// TIA Portal project "Project1" (V16)

(* hardware
DEVICE "S7-1200 station_1"  S7-1200 Station
   slot 0: "Rack_0"  S7-1200 Rack  Rack  V1.0
   slot 1: "PLC_1"  CPU 1214C AC/DC/Rly  6ES7 214-1BG40-0XB0  V4.4
DEVICE "PC-System_1"  SIMATIC PC station
   slot 0: "SIMATIC PC station"  Rail  SIMATIC PC-Station  V1.0
      slot 125: "Stationmanager"  Station_Manager  V6.0.4
   slot 1: "HMI_RT_1"  WinCC RT Advanced  6AV2 104-0xxxx-xxxx  16.0.0.0
      slot 33792: "Computer interface"  Host interface
   slot 2: "IE general_1"  IE General  IE_CP  V8.2.0
*)

// ===== PLC "PLC_1"  CPU 1214C AC/DC/Rly =====

VAR_GLOBAL   // PLC tag table "Default tag table"
   "Tag_1" AT %MW20 : UInt;
   "TIMER_1" AT %MW22 : UInt;
   "TIMER_2" AT %MW24 : UInt;
   "INPUT_X1_INT" AT %MW26 : UInt;
   "INPUT_V1_INT" AT %MW28 : UInt;
   "INPUT_X2_INT" AT %MW30 : UInt;
   "INPUT_V2_INT" AT %MW32 : UInt;
   "INPUT_XV1_INT" AT %MW34 : UInt;
   "INPUT_XV2_INT" AT %MW36 : UInt;
   "INPUT_SUM_INT" AT %MW38 : UInt;
   "INPUT_X1" AT %MD50 : Time;
   "INPUT_V1" AT %MD54 : Time;
   "INPUT_XV1" AT %MD58 : Time;
   "INPUT_X2" AT %MD62 : Time;
   "INPUT_V2" AT %MD66 : Time;
   "INPUT_XV2" AT %MD70 : Time;
   "INPUT_SUM" AT %MD78 : Time;
   "Tag_2" AT %MW100 : UInt;
   "Tag_3" AT %MW102 : UInt;
   "Tag_4" AT %MW104 : UInt;
   "Tag_5" AT %MW106 : UInt;
   "Tag_6" AT %MW108 : UInt;
   "X1_TG" AT %MW200 : UInt;
   "V1_TG" AT %MW202 : UInt;
   "X2_TG" AT %MW204 : UInt;
   "V2_TG" AT %MW206 : UInt;
   "XV1_TG" AT %MW208 : UInt;
   "XV2_TG" AT %MW210 : UInt;
   "XV1X2_TG" AT %MW212 : UInt;
   "INPUT_XV1X2_INT" AT %MW40 : UInt;
   "INPUT_XV1X2" AT %MD74 : Time;
   "SUM_TG" AT %MW214 : UInt;
   "Tag_7" AT %M10.0 : Bool;
   "System_Byte" AT %MB1 : Byte;
   "FirstScan" AT %M1.0 : Bool;
   "DiagStatusUpdate" AT %M1.1 : Bool;
   "AlwaysTRUE" AT %M1.2 : Bool;
   "AlwaysFALSE" AT %M1.3 : Bool;
   "Clock_Byte" AT %MB0 : Byte;
   "Clock_10Hz" AT %M0.0 : Bool;
   "Clock_5Hz" AT %M0.1 : Bool;
   "Clock_2.5Hz" AT %M0.2 : Bool;
   "Clock_2Hz" AT %M0.3 : Bool;
   "Clock_1.25Hz" AT %M0.4 : Bool;
   "Clock_1Hz" AT %M0.5 : Bool;
   "Clock_0.625Hz" AT %M0.6 : Bool;
   "Clock_0.5Hz" AT %M0.7 : Bool;
   "Start" AT %M20.0 : Bool;
   "Stop" AT %M20.1 : Bool;
   "Data" AT %MW70 : Int;
   "Tag_8" AT %MW50 : Int;
   "Tag_9" AT %MD10 : Real;
   "Tag_10" AT %MD14 : Real;
   "He_so_k" AT %MD200 : Real;
   "Tag_11" AT %M50.0 : Bool;
   "Tag_12" AT %M5.0 : Bool;
END_VAR

VAR_GLOBAL   // PLC tag table "Tag table_1"
   "X1_IN" AT %I0.0 : Bool;
   "V1_IN" AT %I0.1 : Bool;
   "X2_IN" AT %I0.2 : Bool;
   "V2_IN" AT %I0.3 : Bool;
   "Bus1" AT %MW82 : Int;
   "Car1" AT %MW84 : Int;
   "Motor1" AT %MW86 : Int;
   "Truck1" AT %MW112 : Int;
   "Bus2" AT %MW90 : Int;
   "Car2" AT %MW92 : Int;
   "Motor2" AT %MW94 : Int;
   "Truck2" AT %MW96 : Int;
   "Sum_h1" AT %MW98 : Int;
   "Sum_h2" AT %MW110 : Int;
END_VAR

DATA_BLOCK "DGT"   // DB1
{ S7_Optimized_Access := 'FALSE' }
VERSION : 0.1
   VAR
      RUN : Bool;
      START : Bool;
      STOP : Bool;
      RED_A : Bool;
      YELLOW_A : Bool;
      GREEN_A : Bool;
      RED_B : Bool;
      YELLOW_B : Bool;
      GREEN_B : Bool;
      AUTO : Bool;
      MAN : Bool;
      SETTING : Bool;
      Q_AUTO : Bool;
      Q_MANU : Bool;
      Q_SETTING : Bool;
   END_VAR
BEGIN
END_DATA_BLOCK

DATA_BLOCK "DB_MANU"   // DB7
{ S7_Optimized_Access := 'TRUE' }
VERSION : 0.1
   VAR
      BT_1 : Bool;
      BT_2 : Bool;
      BT_3 : Bool;
   END_VAR
BEGIN
END_DATA_BLOCK

// folder: System blocks/Program resources

DATA_BLOCK "T1"   // DB2
{ S7_Optimized_Access := 'TRUE' }
AUTHOR : Simatic
FAMILY : IEC
NAME : IEC_TMR
VERSION : 1.0
// stored: InstanceOfName IEC_TIMER
"IEC_TIMER"
BEGIN
END_DATA_BLOCK

// folder: (top level)

FUNCTION "MODE_MANU" : Void   // FC1, LAD
{ S7_Optimized_Access := 'TRUE' }
VERSION : 0.1
BEGIN

REGION Network 1
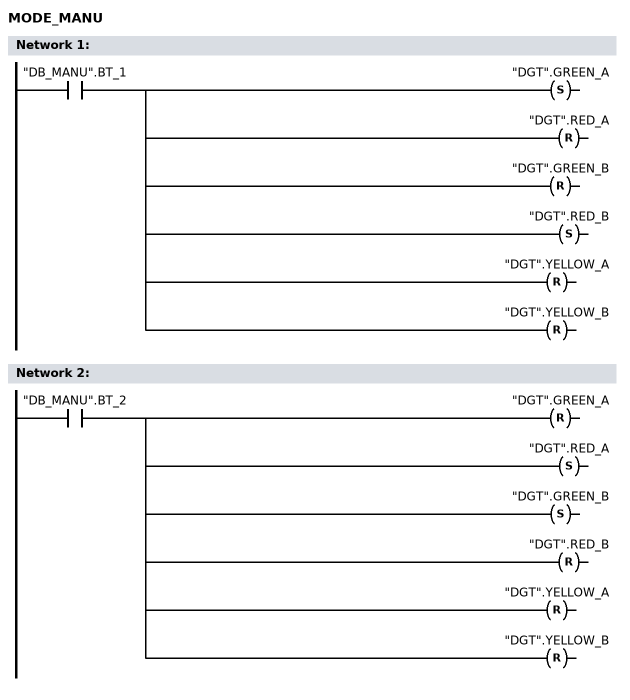
   RUNG wire#powerrail
      Contact( "DB_MANU".BT_1 )
      wire#w1
      S_Coil( "DGT".GREEN_A )
   END_RUNG
   RUNG wire#w1
      R_Coil( "DGT".RED_A )
   END_RUNG
   RUNG wire#w1
      R_Coil( "DGT".GREEN_B )
   END_RUNG
   RUNG wire#w1
      S_Coil( "DGT".RED_B )
   END_RUNG
   RUNG wire#w1
      R_Coil( "DGT".YELLOW_A )
   END_RUNG
   RUNG wire#w1
      R_Coil( "DGT".YELLOW_B )
   END_RUNG
   // the same network as SCL:
   IF "DB_MANU".BT_1 THEN
       "DGT".GREEN_A := TRUE;
       "DGT".RED_A := FALSE;
       "DGT".GREEN_B := FALSE;
       "DGT".RED_B := TRUE;
       "DGT".YELLOW_A := FALSE;
       "DGT".YELLOW_B := FALSE;
   END_IF;
END_REGION

REGION Network 2
   RUNG wire#powerrail
      Contact( "DB_MANU".BT_2 )
      wire#w1
      R_Coil( "DGT".GREEN_A )
   END_RUNG
   RUNG wire#w1
      S_Coil( "DGT".RED_A )
   END_RUNG
   RUNG wire#w1
      S_Coil( "DGT".GREEN_B )
   END_RUNG
   RUNG wire#w1
      R_Coil( "DGT".RED_B )
   END_RUNG
   RUNG wire#w1
      R_Coil( "DGT".YELLOW_A )
   END_RUNG
   RUNG wire#w1
      R_Coil( "DGT".YELLOW_B )
   END_RUNG
   // the same network as SCL:
   IF "DB_MANU".BT_2 THEN
       "DGT".GREEN_A := FALSE;
       "DGT".RED_A := TRUE;
       "DGT".GREEN_B := TRUE;
       "DGT".RED_B := FALSE;
       "DGT".YELLOW_A := FALSE;
       "DGT".YELLOW_B := FALSE;
   END_IF;
END_REGION
END_FUNCTION

FUNCTION "START_UP" : Void   // FC2, LAD
{ S7_Optimized_Access := 'TRUE' }
VERSION : 0.1
BEGIN

REGION Network 1
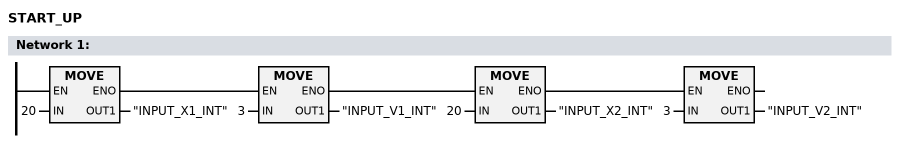
   RUNG wire#powerrail
      Move(in := 20, out1 => "INPUT_X1_INT")
      Move(in := 3, out1 => "INPUT_V1_INT")
      Move(in := 20, out1 => "INPUT_X2_INT")
      Move(in := 3, out1 => "INPUT_V2_INT")
   END_RUNG
   // the same network as SCL:
   "INPUT_X1_INT" := 20;
   "INPUT_V1_INT" := 3;
   "INPUT_X2_INT" := 20;
   "INPUT_V2_INT" := 3;
END_REGION
END_FUNCTION

FUNCTION "MODE_SETTING" : Void   // FC3, LAD
{ S7_Optimized_Access := 'TRUE' }
VERSION : 0.1
   VAR_TEMP   // added for the SCL form of the ladder/FBD networks
      _w1 : Bool;
   END_VAR
BEGIN

REGION Network 1
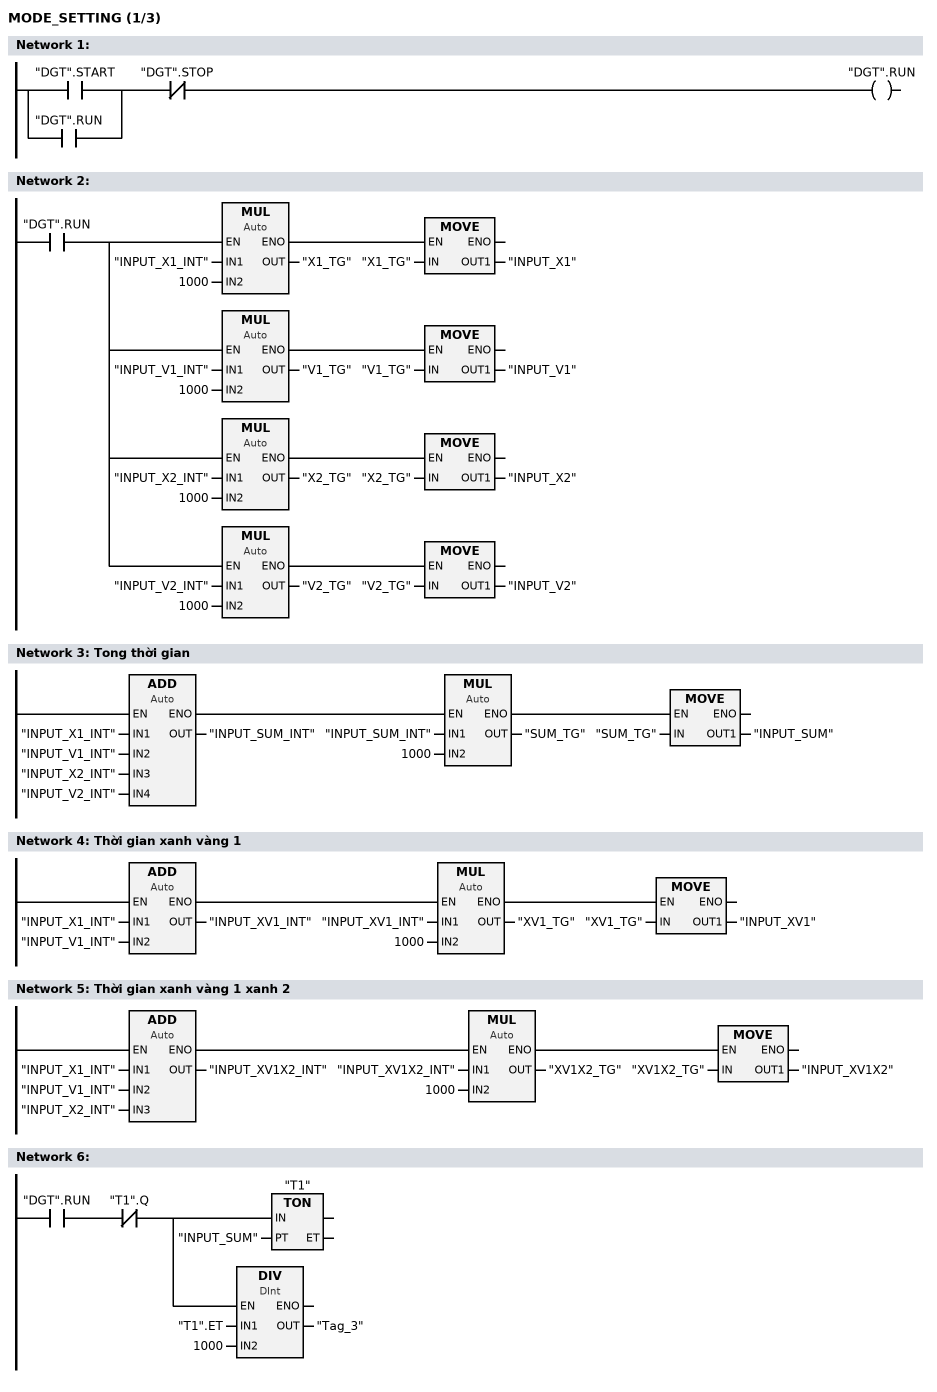
   RUNG wire#powerrail
      Contact( "DGT".START )
      wire#w1
      I_Contact( "DGT".STOP )
      Coil( "DGT".RUN )
   END_RUNG
   RUNG wire#powerrail
      Contact( "DGT".RUN )
   END_RUNG wire#w1
   // the same network as SCL:
   "DGT".RUN := ("DGT".START OR "DGT".RUN) AND NOT "DGT".STOP;
END_REGION

REGION Network 2
   RUNG wire#powerrail
      Contact( "DGT".RUN )
      wire#w1
      Mul(in1 := "INPUT_X1_INT", in2 := 1000, out => "X1_TG")
      Move(in := "X1_TG", out1 => "INPUT_X1")
   END_RUNG
   RUNG wire#w1
      Mul(in1 := "INPUT_V1_INT", in2 := 1000, out => "V1_TG")
      Move(in := "V1_TG", out1 => "INPUT_V1")
   END_RUNG
   RUNG wire#w1
      Mul(in1 := "INPUT_X2_INT", in2 := 1000, out => "X2_TG")
      Move(in := "X2_TG", out1 => "INPUT_X2")
   END_RUNG
   RUNG wire#w1
      Mul(in1 := "INPUT_V2_INT", in2 := 1000, out => "V2_TG")
      Move(in := "V2_TG", out1 => "INPUT_V2")
   END_RUNG
   // the same network as SCL:
   IF "DGT".RUN THEN
       "X1_TG" := "INPUT_X1_INT" * 1000;
       "INPUT_X1" := "X1_TG";
       "V1_TG" := "INPUT_V1_INT" * 1000;
       "INPUT_V1" := "V1_TG";
       "X2_TG" := "INPUT_X2_INT" * 1000;
       "INPUT_X2" := "X2_TG";
       "V2_TG" := "INPUT_V2_INT" * 1000;
       "INPUT_V2" := "V2_TG";
   END_IF;
END_REGION

REGION Network 3: Tong thời gian
   RUNG wire#powerrail
      Add(in1 := "INPUT_X1_INT", in2 := "INPUT_V1_INT", in3 := "INPUT_X2_INT", in4 := "INPUT_V2_INT", out => "INPUT_SUM_INT")
      Mul(in1 := "INPUT_SUM_INT", in2 := 1000, out => "SUM_TG")
      Move(in := "SUM_TG", out1 => "INPUT_SUM")
   END_RUNG
   // the same network as SCL:
   "INPUT_SUM_INT" := "INPUT_X1_INT" + "INPUT_V1_INT" + "INPUT_X2_INT" + "INPUT_V2_INT";
   "SUM_TG" := "INPUT_SUM_INT" * 1000;
   "INPUT_SUM" := "SUM_TG";
END_REGION

REGION Network 4: Thời gian xanh vàng 1
   RUNG wire#powerrail
      Add(in1 := "INPUT_X1_INT", in2 := "INPUT_V1_INT", out => "INPUT_XV1_INT")
      Mul(in1 := "INPUT_XV1_INT", in2 := 1000, out => "XV1_TG")
      Move(in := "XV1_TG", out1 => "INPUT_XV1")
   END_RUNG
   // the same network as SCL:
   "INPUT_XV1_INT" := "INPUT_X1_INT" + "INPUT_V1_INT";
   "XV1_TG" := "INPUT_XV1_INT" * 1000;
   "INPUT_XV1" := "XV1_TG";
END_REGION

REGION Network 5: Thời gian xanh vàng 1 xanh 2
   RUNG wire#powerrail
      Add(in1 := "INPUT_X1_INT", in2 := "INPUT_V1_INT", in3 := "INPUT_X2_INT", out => "INPUT_XV1X2_INT")
      Mul(in1 := "INPUT_XV1X2_INT", in2 := 1000, out => "XV1X2_TG")
      Move(in := "XV1X2_TG", out1 => "INPUT_XV1X2")
   END_RUNG
   // the same network as SCL:
   "INPUT_XV1X2_INT" := "INPUT_X1_INT" + "INPUT_V1_INT" + "INPUT_X2_INT";
   "XV1X2_TG" := "INPUT_XV1X2_INT" * 1000;
   "INPUT_XV1X2" := "XV1X2_TG";
END_REGION

REGION Network 6
   #_w1 := "DGT".RUN AND NOT "T1".Q;
   "T1".TON(IN := #_w1, PT := "INPUT_SUM");
   IF #_w1 THEN "Tag_3" := "T1".ET / 1000; END_IF;
END_REGION

REGION Network 7
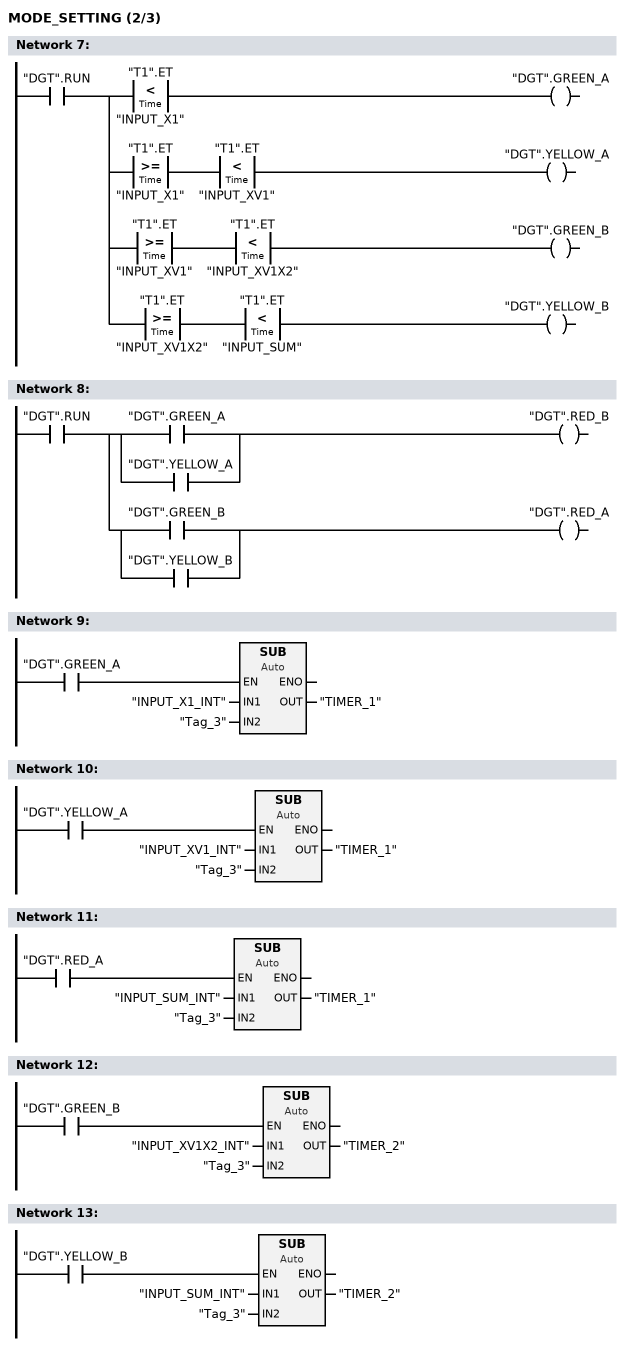
   RUNG wire#powerrail
      Contact( "DGT".RUN )
      wire#w1
      { S7_Templates := "SrcType := Time" } LT_Contact(in1 := "T1".ET, in2 := "INPUT_X1")
      Coil( "DGT".GREEN_A )
   END_RUNG
   RUNG wire#w1
      { S7_Templates := "SrcType := Time" } GE_Contact(in1 := "T1".ET, in2 := "INPUT_X1")
      { S7_Templates := "SrcType := Time" } LT_Contact(in1 := "T1".ET, in2 := "INPUT_XV1")
      Coil( "DGT".YELLOW_A )
   END_RUNG
   RUNG wire#w1
      { S7_Templates := "SrcType := Time" } GE_Contact(in1 := "T1".ET, in2 := "INPUT_XV1")
      { S7_Templates := "SrcType := Time" } LT_Contact(in1 := "T1".ET, in2 := "INPUT_XV1X2")
      Coil( "DGT".GREEN_B )
   END_RUNG
   RUNG wire#w1
      { S7_Templates := "SrcType := Time" } GE_Contact(in1 := "T1".ET, in2 := "INPUT_XV1X2")
      { S7_Templates := "SrcType := Time" } LT_Contact(in1 := "T1".ET, in2 := "INPUT_SUM")
      Coil( "DGT".YELLOW_B )
   END_RUNG
   // the same network as SCL:
   "DGT".GREEN_A := "DGT".RUN AND ("T1".ET < "INPUT_X1");
   "DGT".YELLOW_A := "DGT".RUN AND ("T1".ET >= "INPUT_X1") AND ("T1".ET < "INPUT_XV1");
   "DGT".GREEN_B := "DGT".RUN AND ("T1".ET >= "INPUT_XV1") AND ("T1".ET < "INPUT_XV1X2");
   "DGT".YELLOW_B := "DGT".RUN AND ("T1".ET >= "INPUT_XV1X2") AND ("T1".ET < "INPUT_SUM");
END_REGION

REGION Network 8
   RUNG wire#powerrail
      Contact( "DGT".RUN )
      wire#w1
      Contact( "DGT".GREEN_A )
      wire#w2
      Coil( "DGT".RED_B )
   END_RUNG
   RUNG wire#w1
      Contact( "DGT".YELLOW_A )
   END_RUNG wire#w2
   RUNG wire#w1
      Contact( "DGT".GREEN_B )
      wire#w3
      Coil( "DGT".RED_A )
   END_RUNG
   RUNG wire#w1
      Contact( "DGT".YELLOW_B )
   END_RUNG wire#w3
   // the same network as SCL:
   "DGT".RED_B := "DGT".RUN AND ("DGT".GREEN_A OR "DGT".YELLOW_A);
   "DGT".RED_A := "DGT".RUN AND ("DGT".GREEN_B OR "DGT".YELLOW_B);
END_REGION

REGION Network 9
   RUNG wire#powerrail
      Contact( "DGT".GREEN_A )
      Sub(in1 := "INPUT_X1_INT", in2 := "Tag_3", out => "TIMER_1")
   END_RUNG
   // the same network as SCL:
   IF "DGT".GREEN_A THEN "TIMER_1" := "INPUT_X1_INT" - "Tag_3"; END_IF;
END_REGION

REGION Network 10
   RUNG wire#powerrail
      Contact( "DGT".YELLOW_A )
      Sub(in1 := "INPUT_XV1_INT", in2 := "Tag_3", out => "TIMER_1")
   END_RUNG
   // the same network as SCL:
   IF "DGT".YELLOW_A THEN "TIMER_1" := "INPUT_XV1_INT" - "Tag_3"; END_IF;
END_REGION

REGION Network 11
   RUNG wire#powerrail
      Contact( "DGT".RED_A )
      Sub(in1 := "INPUT_SUM_INT", in2 := "Tag_3", out => "TIMER_1")
   END_RUNG
   // the same network as SCL:
   IF "DGT".RED_A THEN "TIMER_1" := "INPUT_SUM_INT" - "Tag_3"; END_IF;
END_REGION

REGION Network 12
   RUNG wire#powerrail
      Contact( "DGT".GREEN_B )
      Sub(in1 := "INPUT_XV1X2_INT", in2 := "Tag_3", out => "TIMER_2")
   END_RUNG
   // the same network as SCL:
   IF "DGT".GREEN_B THEN "TIMER_2" := "INPUT_XV1X2_INT" - "Tag_3"; END_IF;
END_REGION

REGION Network 13
   RUNG wire#powerrail
      Contact( "DGT".YELLOW_B )
      Sub(in1 := "INPUT_SUM_INT", in2 := "Tag_3", out => "TIMER_2")
   END_RUNG
   // the same network as SCL:
   IF "DGT".YELLOW_B THEN "TIMER_2" := "INPUT_SUM_INT" - "Tag_3"; END_IF;
END_REGION

REGION Network 14
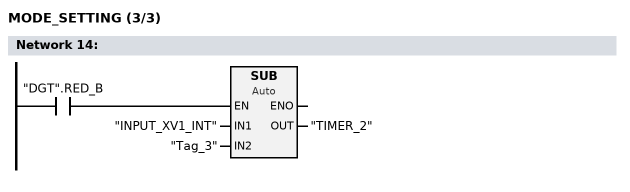
   RUNG wire#powerrail
      Contact( "DGT".RED_B )
      Sub(in1 := "INPUT_XV1_INT", in2 := "Tag_3", out => "TIMER_2")
   END_RUNG
   // the same network as SCL:
   IF "DGT".RED_B THEN "TIMER_2" := "INPUT_XV1_INT" - "Tag_3"; END_IF;
END_REGION
END_FUNCTION

FUNCTION "BROKER" : Void   // FC4, LAD
{ S7_Optimized_Access := 'TRUE' }
VERSION : 0.1
BEGIN

REGION Network 1
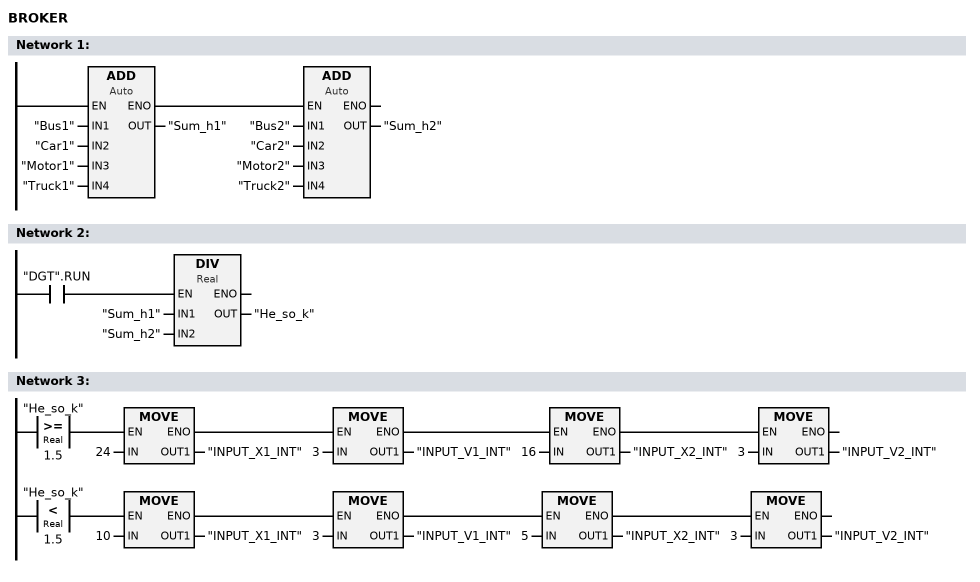
   RUNG wire#powerrail
      Add(in1 := "Bus1", in2 := "Car1", in3 := "Motor1", in4 := "Truck1", out => "Sum_h1")
      Add(in1 := "Bus2", in2 := "Car2", in3 := "Motor2", in4 := "Truck2", out => "Sum_h2")
   END_RUNG
   // the same network as SCL:
   "Sum_h1" := "Bus1" + "Car1" + "Motor1" + "Truck1";
   "Sum_h2" := "Bus2" + "Car2" + "Motor2" + "Truck2";
END_REGION

REGION Network 2
   RUNG wire#powerrail
      Contact( "DGT".RUN )
      { S7_Templates := "SrcType := Real" } Div(in1 := "Sum_h1", in2 := "Sum_h2", out => "He_so_k")
   END_RUNG
   // the same network as SCL:
   IF "DGT".RUN THEN "He_so_k" := "Sum_h1" / "Sum_h2"; END_IF;
END_REGION

REGION Network 3
   RUNG wire#powerrail
      { S7_Templates := "SrcType := Real" } GE_Contact(in1 := "He_so_k", in2 := 1.5)
      Move(in := 24, out1 => "INPUT_X1_INT")
      Move(in := 3, out1 => "INPUT_V1_INT")
      Move(in := 16, out1 => "INPUT_X2_INT")
      Move(in := 3, out1 => "INPUT_V2_INT")
   END_RUNG
   RUNG wire#powerrail
      { S7_Templates := "SrcType := Real" } LT_Contact(in1 := "He_so_k", in2 := 1.5)
      Move(in := 10, out1 => "INPUT_X1_INT")
      Move(in := 3, out1 => "INPUT_V1_INT")
      Move(in := 5, out1 => "INPUT_X2_INT")
      Move(in := 3, out1 => "INPUT_V2_INT")
   END_RUNG
   // the same network as SCL:
   IF "He_so_k" >= 1.5 THEN
       "INPUT_X1_INT" := 24;
       "INPUT_V1_INT" := 3;
       "INPUT_X2_INT" := 16;
       "INPUT_V2_INT" := 3;
   END_IF;
   IF "He_so_k" < 1.5 THEN
       "INPUT_X1_INT" := 10;
       "INPUT_V1_INT" := 3;
       "INPUT_X2_INT" := 5;
       "INPUT_V2_INT" := 3;
   END_IF;
END_REGION
END_FUNCTION

ORGANIZATION_BLOCK "Main"   // OB1, LAD, ProgramCycle
TITLE = "Main Program Sweep (Cycle)"
{ S7_Optimized_Access := 'TRUE' }
VERSION : 0.1
   VAR_INPUT
      Initial_Call : Bool;   // Initial call of this OB
      Remanence : Bool;   // =True, if remanent data are available
   END_VAR
   VAR_TEMP   // added for the SCL form of the ladder/FBD networks
      _w1 : Bool;
   END_VAR
BEGIN

REGION Network 1
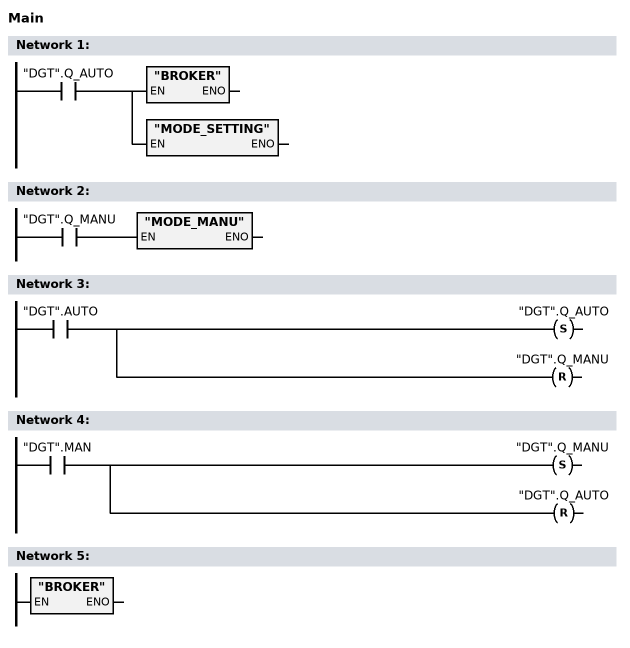
   RUNG wire#powerrail
      Contact( "DGT".Q_AUTO )
      wire#w1
      "BROKER"()
   END_RUNG
   RUNG wire#w1
      "MODE_SETTING"()
   END_RUNG
   // the same network as SCL:
   #_w1 := "DGT".Q_AUTO;
   IF #_w1 THEN
       "BROKER"();
       "MODE_SETTING"();
   END_IF;
END_REGION

REGION Network 2
   RUNG wire#powerrail
      Contact( "DGT".Q_MANU )
      "MODE_MANU"()
   END_RUNG
   // the same network as SCL:
   IF "DGT".Q_MANU THEN "MODE_MANU"(); END_IF;
END_REGION

REGION Network 3
   RUNG wire#powerrail
      Contact( "DGT".AUTO )
      wire#w1
      S_Coil( "DGT".Q_AUTO )
   END_RUNG
   RUNG wire#w1
      R_Coil( "DGT".Q_MANU )
   END_RUNG
   // the same network as SCL:
   IF "DGT".AUTO THEN
       "DGT".Q_AUTO := TRUE;
       "DGT".Q_MANU := FALSE;
   END_IF;
END_REGION

REGION Network 4
   RUNG wire#powerrail
      Contact( "DGT".MAN )
      wire#w1
      S_Coil( "DGT".Q_MANU )
   END_RUNG
   RUNG wire#w1
      R_Coil( "DGT".Q_AUTO )
   END_RUNG
   // the same network as SCL:
   IF "DGT".MAN THEN
       "DGT".Q_MANU := TRUE;
       "DGT".Q_AUTO := FALSE;
   END_IF;
END_REGION

REGION Network 5
   RUNG wire#powerrail
      "BROKER"()
   END_RUNG
   // the same network as SCL:
   "BROKER"();
END_REGION
END_ORGANIZATION_BLOCK

(* ===== HMI "HMI_RT_1" =====
system functions are stored by id; their names below are inferred from use
connection "HMI_Connection_1": ETHERNET, S7_1200_OMS

HMI tags "Default tag table"
   "DGT_XANH_A" : Bool = PLC DGT.GREEN_A AT %DB1.DBX0.5, 1 s
   "DGT_VANG_A" : Bool = PLC DGT.YELLOW_A AT %DB1.DBX0.4, 1 s
   "DGT_DO_A" : Bool = PLC DGT.RED_A AT %DB1.DBX0.3, 1 s
   "INPUT_X1_INT" : UInt = PLC INPUT_X1_INT AT %MW26, 100 ms
   "INPUT_V1_INT" : UInt = PLC INPUT_V1_INT AT %MW28, 100 ms
   "INPUT_X2_INT" : UInt = PLC INPUT_X2_INT AT %MW30, 100 ms
   "INPUT_V2_INT" : UInt = PLC INPUT_V2_INT AT %MW32, 100 ms
   "DGT_START" : Bool = PLC DGT.START AT %DB1.DBX0.1, 100 ms
   "DGT_AUTO" : Bool = PLC DGT.AUTO AT %DB1.DBX1.1, 100 ms
   "DGT_STOP" : Bool = PLC DGT.STOP AT %DB1.DBX0.2, 100 ms
   "DGT_VANG_B" : Bool = PLC DGT.YELLOW_B AT %DB1.DBX0.7, 1 s
   "DGT_XANH_B" : Bool = PLC DGT.GREEN_B AT %DB1.DBX1.0, 1 s
   "DGT_DO_B" : Bool = PLC DGT.RED_B AT %DB1.DBX0.6, 1 s
   "TIMER_1" : UInt = PLC TIMER_1 AT %MW22, 1 s
   "TIMER_2" : UInt = PLC TIMER_2 AT %MW24, 1 s
   "DB_MANU_BT_1" : Bool = PLC DB_MANU.BT_1, 100 ms
   "DB_MANU_BT_2" : Bool = PLC DB_MANU.BT_2, 100 ms
   "DB_MANU_BT_3" : Bool = PLC DB_MANU.BT_3, 100 ms
   "DGT_SETTING" : Bool = PLC DGT.SETTING AT %DB1.DBX1.3, 100 ms
   "DGT_MAN" : Bool = PLC DGT.MAN AT %DB1.DBX1.2, 100 ms
   "Sum_h1" : Int = PLC Sum_h1 AT %MW98, 1 s
   "Sum_h2" : Int = PLC Sum_h2 AT %MW110, 1 s

screen "Screen_1" 1024x768
   IOField "I/O field_1" at 78,191 size 84x33; FormatPattern 99999
      ProcessValue <- "INPUT_X1_INT"
   IOField "I/O field_2" at 78,231 size 84x33; FormatPattern 99999
      ProcessValue <- "INPUT_V1_INT"
   IOField "I/O field_3" at 78,271 size 84x33; FormatPattern 99999
      ProcessValue <- "INPUT_X2_INT"
   IOField "I/O field_4" at 78,311 size 84x33; FormatPattern 99999
      ProcessValue <- "INPUT_V2_INT"
   Button "Button_1" at 132,75 size 83x36; TextOff 'START'
      on Press: SetBit("DGT_START")
      on Release: ResetBit("DGT_START")
   Button "Button_2" at 130,127 size 85x35; TextOff 'STOP'
      on Press: SetBit("DGT_STOP")
      on Release: ResetBit("DGT_STOP")
   Button "Button_3" at 18,83 size 78x31; TextOff 'LINE 1'
      on Press: SetBit("DB_MANU_BT_1")
      on Release: ResetBit("DB_MANU_BT_1")
   Button "Button_4" at 18,130 size 78x31; TextOff 'LINE 2'
      on Press: SetBit("DB_MANU_BT_2")
      on Release: ResetBit("DB_MANU_BT_2")
   TextField "Text field_1" at 5,197 size 62x22; Text 'XANH 1'
   TextField "Text field_2" at 5,239 size 62x22; Text 'VANG 1'
   TextField "Text field_3" at 5,276 size 62x22; Text 'XANH 1'
   TextField "Text field_4" at 7,315 size 62x22; Text 'VANG 2'
   Button "Button_6" at -1,21 size 64x36; TextOff 'MAN'
      on Release: ResetBit("DGT_MAN")
      on Press: SetBit("DGT_MAN")
   Button "Button_7" at 71,21 size 64x36; TextOff 'AUTO'
      on Release: ResetBit("DGT_AUTO")
      on Press: SetBit("DGT_AUTO")
   TextField "Text field_5" at 716,70 size 56x22; Text 'LINE 1'
   Circle "Circle_1" at 686,459 size 35x35
      Appearance <- "DGT_DO_A"
   Circle "Circle_2" at 686,494 size 35x35
      Appearance <- "DGT_VANG_A"
   Circle "Circle_3" at 686,529 size 35x35
      Appearance <- "DGT_XANH_A"
   Circle "Circle_4" at 490,185 size 35x35
      Appearance <- "DGT_XANH_A"
   Circle "Circle_5" at 490,220 size 35x35
      Appearance <- "DGT_VANG_A"
   Circle "Circle_6" at 490,255 size 35x35
      Appearance <- "DGT_DO_A"
   Circle "Circle_7" at 686,255 size 35x35
      Appearance <- "DGT_DO_B"
   Circle "Circle_8" at 721,255 size 35x35
      Appearance <- "DGT_VANG_B"
   Circle "Circle_9" at 756,255 size 35x35
      Appearance <- "DGT_XANH_B"
   Circle "Circle_10" at 491,450 size 35x35
      Appearance <- "DGT_DO_B"
   Circle "Circle_11" at 456,450 size 35x35
      Appearance <- "DGT_VANG_B"
   Circle "Circle_12" at 421,450 size 35x35
      Appearance <- "DGT_XANH_B"
   IOField "I/O field_5" at 688,421 size 31x31; FormatPattern 99
      ProcessValue <- "TIMER_1"
   IOField "I/O field_6" at 491,297 size 31x31; FormatPattern 99
      ProcessValue <- "TIMER_1"
   IOField "I/O field_8" at 534,453 size 28x32; FormatPattern 99
      ProcessValue <- "TIMER_2"
   SymbolLibrary "Symbol library_1" at 578,311 size 81x28
   SymbolLibrary "Symbol library_2" at 622,142 size 37x62
   SymbolLibrary "Symbol library_3" at 398,387 size 78x23
   IOField "I/O field_7" at 649,256 size 28x32; FormatPattern 99
      ProcessValue <- "TIMER_2"
   SymbolLibrary "Symbol library_4" at 815,244 size 39x44
   SymbolLibrary "Symbol library_5" at 907,251 size 22x37
   SymbolLibrary "Symbol library_6" at 775,411 size 33x38
   SymbolLibrary "Symbol library_7" at 873,410 size 33x38
   SymbolLibrary "Symbol library_8" at 374,412 size 33x38
   SymbolLibrary "Symbol library_9" at 291,411 size 33x38
   SymbolLibrary "Symbol library_10" at 402,252 size 19x38
   SymbolLibrary "Symbol library_11" at 274,252 size 28x38
   SymbolLibrary "Symbol library_12" at 343,251 size 19x38
*)